// TIA Portal V18 export
FUNCTION_BLOCK "Baustein_1"   // FB1, FBD
{ S7_Optimized_Access := 'TRUE' }
// stored: MemoryReserve 100, SetENOAutomatically false
   VAR_OUTPUT
      Input_1 : Bool;
      Input_2 : Int := 200;
      Input_3 : Int := 2001;
   END_VAR
BEGIN

REGION Network 1
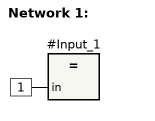
   #Input_1 := 1;
END_REGION
END_FUNCTION_BLOCK
